Fanuc KAREL source: tst_csv_writ.kl

PROGRAM tst_csv_writ
%NOLOCKGROUP

VAR
  block_write FROM tst_csv_main : INTEGER
  entries FROM tst_csv_main : INTEGER
  waitime FROM tst_csv_main : INTEGER
  writedelay FROM tst_csv_main  : INTEGER
  pose : XYZWPR
  i, tme : INTEGER
  time_out : BOOLEAN

%include math.klh
%include csv.klh

-- sensor csv file
%class csvpip('csvclass.klc','csvclass.klh')


BEGIN

  FOR i=1 TO entries DO
    --wait for writing to display to finish
    --before continuing to write
    PEND_SEMA(block_write, waitime, time_out)
    IF time_out THEN
      GOTO ENDWRIT
    ENDIF
    --create random initial position
    tme = GET_USEC_TIM
    pose = math__rand_position(tme)
    --write pose to csv pipe
    csvpip__write_row_xyzwpr(pose)

    POST_SEMA (block_write)

    -- create fake work
    DELAY writedelay
  ENDFOR
  -- write to display for remainder data
  csvpip__write_display
  csvpip__clear

  ENDWRIT::
  WRITE TPDISPLAY(CR,'csv write is done.')

END tst_csv_writ
